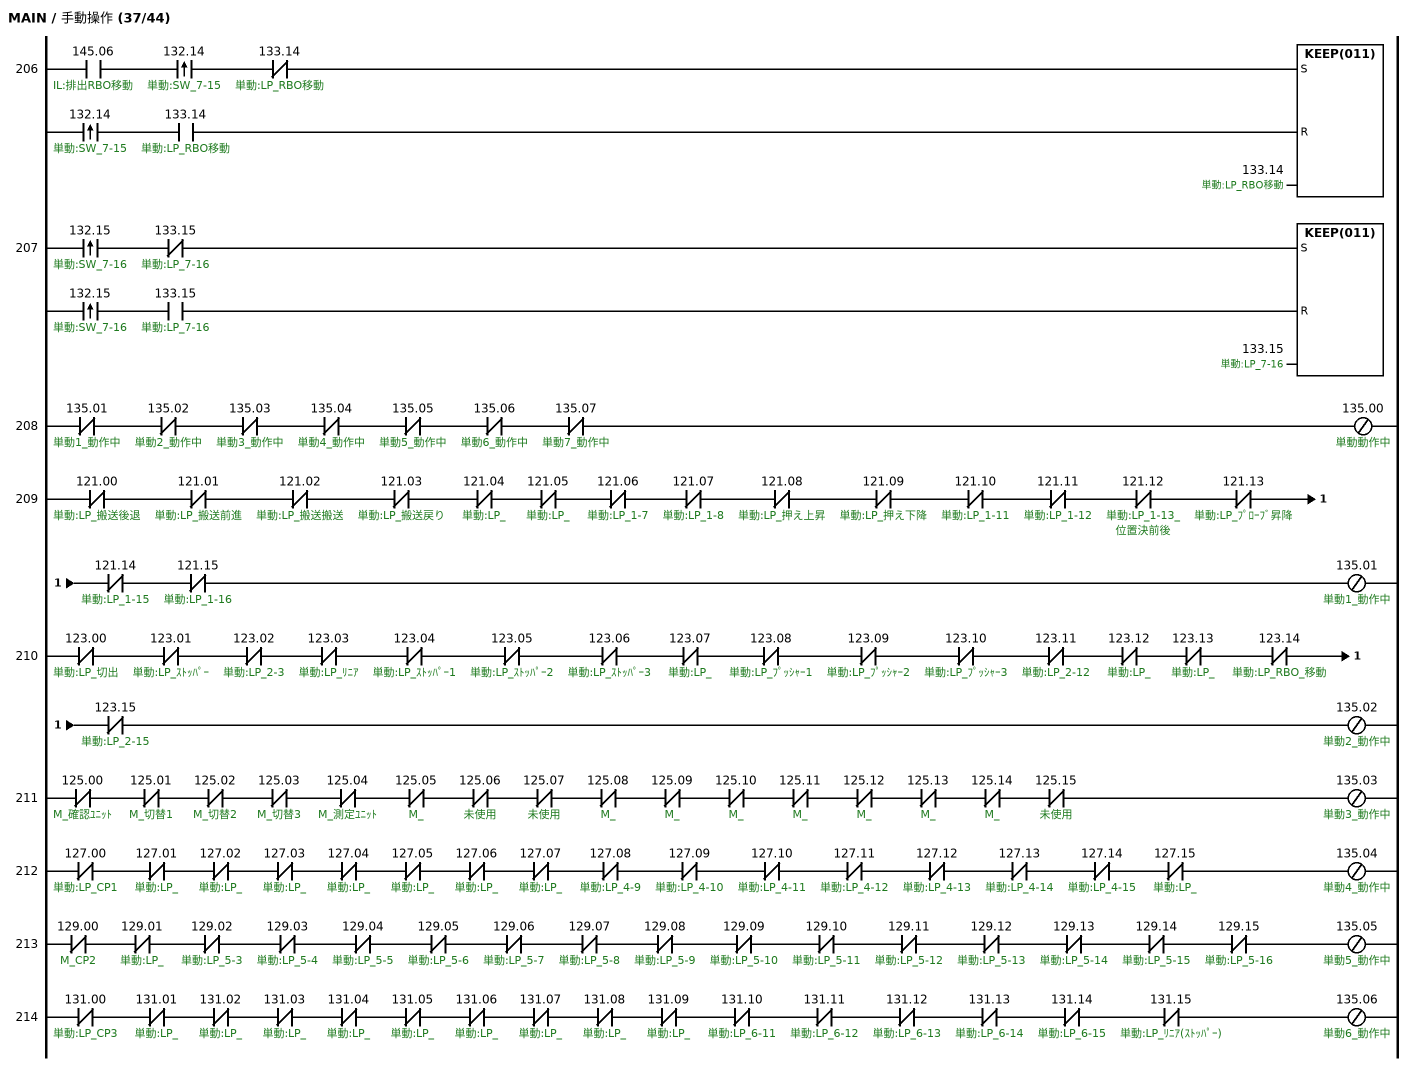
; [picture p72: MAIN / 手動操作, rungs 206-214]
; rung 206
LD 145.06  ; IL:排出RBO移動
@AND 132.14  ; 単動:SW_7-15
ANDNOT 133.14  ; 単動:LP_RBO移動
@LD 132.14  ; 単動:SW_7-15
AND 133.14  ; 単動:LP_RBO移動
KEEP(011) 133.14  ; 単動:LP_RBO移動
; rung 207
@LD 132.15  ; 単動:SW_7-16
ANDNOT 133.15  ; 単動:LP_7-16
@LD 132.15  ; 単動:SW_7-16
AND 133.15  ; 単動:LP_7-16
KEEP(011) 133.15  ; 単動:LP_7-16
; rung 208
LDNOT 135.01  ; 単動1_動作中
ANDNOT 135.02  ; 単動2_動作中
ANDNOT 135.03  ; 単動3_動作中
ANDNOT 135.04  ; 単動4_動作中
ANDNOT 135.05  ; 単動5_動作中
ANDNOT 135.06  ; 単動6_動作中
ANDNOT 135.07  ; 単動7_動作中
OUTNOT 135.00  ; 単動動作中
; rung 209
LDNOT 121.00  ; 単動:LP_搬送後退
ANDNOT 121.01  ; 単動:LP_搬送前進
ANDNOT 121.02  ; 単動:LP_搬送搬送
ANDNOT 121.03  ; 単動:LP_搬送戻り
ANDNOT 121.04  ; 単動:LP_
ANDNOT 121.05  ; 単動:LP_
ANDNOT 121.06  ; 単動:LP_1-7
ANDNOT 121.07  ; 単動:LP_1-8
ANDNOT 121.08  ; 単動:LP_押え上昇
ANDNOT 121.09  ; 単動:LP_押え下降
ANDNOT 121.10  ; 単動:LP_1-11
ANDNOT 121.11  ; 単動:LP_1-12
ANDNOT 121.12  ; 単動:LP_1-13_位置決前後
ANDNOT 121.13  ; 単動:LP_ﾌﾟﾛｰﾌﾞ昇降
ANDNOT 121.14  ; 単動:LP_1-15
ANDNOT 121.15  ; 単動:LP_1-16
OUTNOT 135.01  ; 単動1_動作中
; rung 210
LDNOT 123.00  ; 単動:LP_切出
ANDNOT 123.01  ; 単動:LP_ｽﾄｯﾊﾟｰ
ANDNOT 123.02  ; 単動:LP_2-3
ANDNOT 123.03  ; 単動:LP_ﾘﾆｱ
ANDNOT 123.04  ; 単動:LP_ｽﾄｯﾊﾟｰ1
ANDNOT 123.05  ; 単動:LP_ｽﾄｯﾊﾟｰ2
ANDNOT 123.06  ; 単動:LP_ｽﾄｯﾊﾟｰ3
ANDNOT 123.07  ; 単動:LP_
ANDNOT 123.08  ; 単動:LP_ﾌﾟｯｼｬｰ1
ANDNOT 123.09  ; 単動:LP_ﾌﾟｯｼｬｰ2
ANDNOT 123.10  ; 単動:LP_ﾌﾟｯｼｬｰ3
ANDNOT 123.11  ; 単動:LP_2-12
ANDNOT 123.12  ; 単動:LP_
ANDNOT 123.13  ; 単動:LP_
ANDNOT 123.14  ; 単動:LP_RBO_移動
ANDNOT 123.15  ; 単動:LP_2-15
OUTNOT 135.02  ; 単動2_動作中
; rung 211
LDNOT 125.00  ; M_確認ﾕﾆｯﾄ
ANDNOT 125.01  ; M_切替1
ANDNOT 125.02  ; M_切替2
ANDNOT 125.03  ; M_切替3
ANDNOT 125.04  ; M_測定ﾕﾆｯﾄ
ANDNOT 125.05  ; M_
ANDNOT 125.06  ; 未使用
ANDNOT 125.07  ; 未使用
ANDNOT 125.08  ; M_
ANDNOT 125.09  ; M_
ANDNOT 125.10  ; M_
ANDNOT 125.11  ; M_
ANDNOT 125.12  ; M_
ANDNOT 125.13  ; M_
ANDNOT 125.14  ; M_
ANDNOT 125.15  ; 未使用
OUTNOT 135.03  ; 単動3_動作中
; rung 212
LDNOT 127.00  ; 単動:LP_CP1
ANDNOT 127.01  ; 単動:LP_
ANDNOT 127.02  ; 単動:LP_
ANDNOT 127.03  ; 単動:LP_
ANDNOT 127.04  ; 単動:LP_
ANDNOT 127.05  ; 単動:LP_
ANDNOT 127.06  ; 単動:LP_
ANDNOT 127.07  ; 単動:LP_
ANDNOT 127.08  ; 単動:LP_4-9
ANDNOT 127.09  ; 単動:LP_4-10
ANDNOT 127.10  ; 単動:LP_4-11
ANDNOT 127.11  ; 単動:LP_4-12
ANDNOT 127.12  ; 単動:LP_4-13
ANDNOT 127.13  ; 単動:LP_4-14
ANDNOT 127.14  ; 単動:LP_4-15
ANDNOT 127.15  ; 単動:LP_
OUTNOT 135.04  ; 単動4_動作中
; rung 213
LDNOT 129.00  ; M_CP2
ANDNOT 129.01  ; 単動:LP_
ANDNOT 129.02  ; 単動:LP_5-3
ANDNOT 129.03  ; 単動:LP_5-4
ANDNOT 129.04  ; 単動:LP_5-5
ANDNOT 129.05  ; 単動:LP_5-6
ANDNOT 129.06  ; 単動:LP_5-7
ANDNOT 129.07  ; 単動:LP_5-8
ANDNOT 129.08  ; 単動:LP_5-9
ANDNOT 129.09  ; 単動:LP_5-10
ANDNOT 129.10  ; 単動:LP_5-11
ANDNOT 129.11  ; 単動:LP_5-12
ANDNOT 129.12  ; 単動:LP_5-13
ANDNOT 129.13  ; 単動:LP_5-14
ANDNOT 129.14  ; 単動:LP_5-15
ANDNOT 129.15  ; 単動:LP_5-16
OUTNOT 135.05  ; 単動5_動作中
; rung 214
LDNOT 131.00  ; 単動:LP_CP3
ANDNOT 131.01  ; 単動:LP_
ANDNOT 131.02  ; 単動:LP_
ANDNOT 131.03  ; 単動:LP_
ANDNOT 131.04  ; 単動:LP_
ANDNOT 131.05  ; 単動:LP_
ANDNOT 131.06  ; 単動:LP_
ANDNOT 131.07  ; 単動:LP_
ANDNOT 131.08  ; 単動:LP_
ANDNOT 131.09  ; 単動:LP_
ANDNOT 131.10  ; 単動:LP_6-11
ANDNOT 131.11  ; 単動:LP_6-12
ANDNOT 131.12  ; 単動:LP_6-13
ANDNOT 131.13  ; 単動:LP_6-14
ANDNOT 131.14  ; 単動:LP_6-15
ANDNOT 131.15  ; 単動:LP_ﾘﾆｱ(ｽﾄｯﾊﾟｰ)
OUTNOT 135.06  ; 単動6_動作中

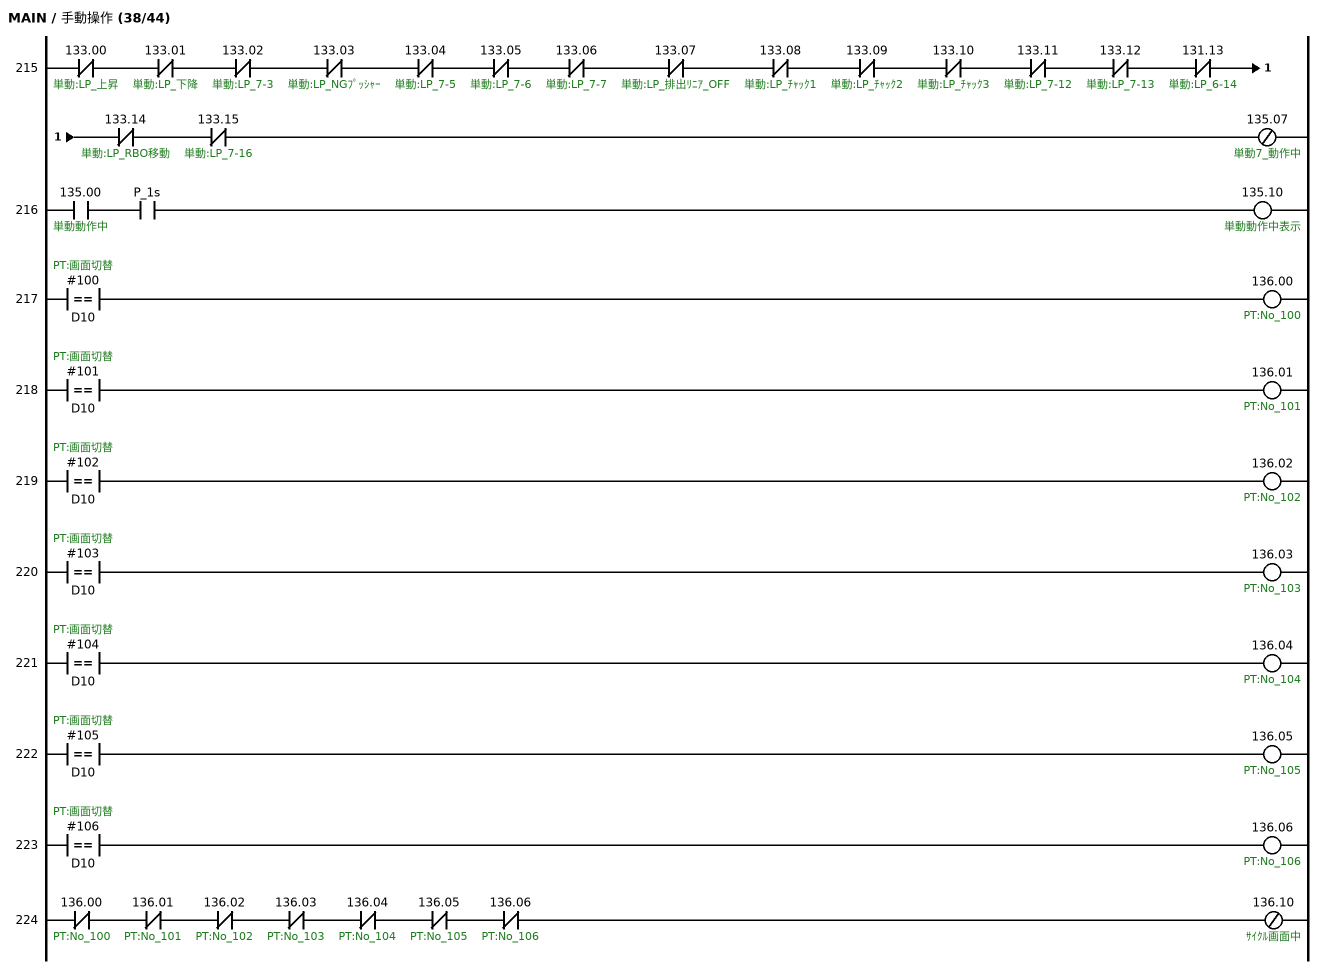
; rung 215
LDNOT 133.00  ; 単動:LP_上昇
ANDNOT 133.01  ; 単動:LP_下降
ANDNOT 133.02  ; 単動:LP_7-3
ANDNOT 133.03  ; 単動:LP_NGﾌﾟｯｼｬｰ
ANDNOT 133.04  ; 単動:LP_7-5
ANDNOT 133.05  ; 単動:LP_7-6
ANDNOT 133.06  ; 単動:LP_7-7
ANDNOT 133.07  ; 単動:LP_排出ﾘﾆｱ_OFF
ANDNOT 133.08  ; 単動:LP_ﾁｬｯｸ1
ANDNOT 133.09  ; 単動:LP_ﾁｬｯｸ2
ANDNOT 133.10  ; 単動:LP_ﾁｬｯｸ3
ANDNOT 133.11  ; 単動:LP_7-12
ANDNOT 133.12  ; 単動:LP_7-13
ANDNOT 131.13  ; 単動:LP_6-14
ANDNOT 133.14  ; 単動:LP_RBO移動
ANDNOT 133.15  ; 単動:LP_7-16
OUTNOT 135.07  ; 単動7_動作中
; rung 216
LD 135.00  ; 単動動作中
AND P_1s
OUT 135.10  ; 単動動作中表示
; rung 217
LD=(300) #100 D10  ; PT:画面切替
OUT 136.00  ; PT:No_100
; rung 218
LD=(300) #101 D10  ; PT:画面切替
OUT 136.01  ; PT:No_101
; rung 219
LD=(300) #102 D10  ; PT:画面切替
OUT 136.02  ; PT:No_102
; rung 220
LD=(300) #103 D10  ; PT:画面切替
OUT 136.03  ; PT:No_103
; rung 221
LD=(300) #104 D10  ; PT:画面切替
OUT 136.04  ; PT:No_104
; rung 222
LD=(300) #105 D10  ; PT:画面切替
OUT 136.05  ; PT:No_105
; rung 223
LD=(300) #106 D10  ; PT:画面切替
OUT 136.06  ; PT:No_106
; rung 224
LDNOT 136.00  ; PT:No_100
ANDNOT 136.01  ; PT:No_101
ANDNOT 136.02  ; PT:No_102
ANDNOT 136.03  ; PT:No_103
ANDNOT 136.04  ; PT:No_104
ANDNOT 136.05  ; PT:No_105
ANDNOT 136.06  ; PT:No_106
OUTNOT 136.10  ; ｻｲｸﾙ画面中

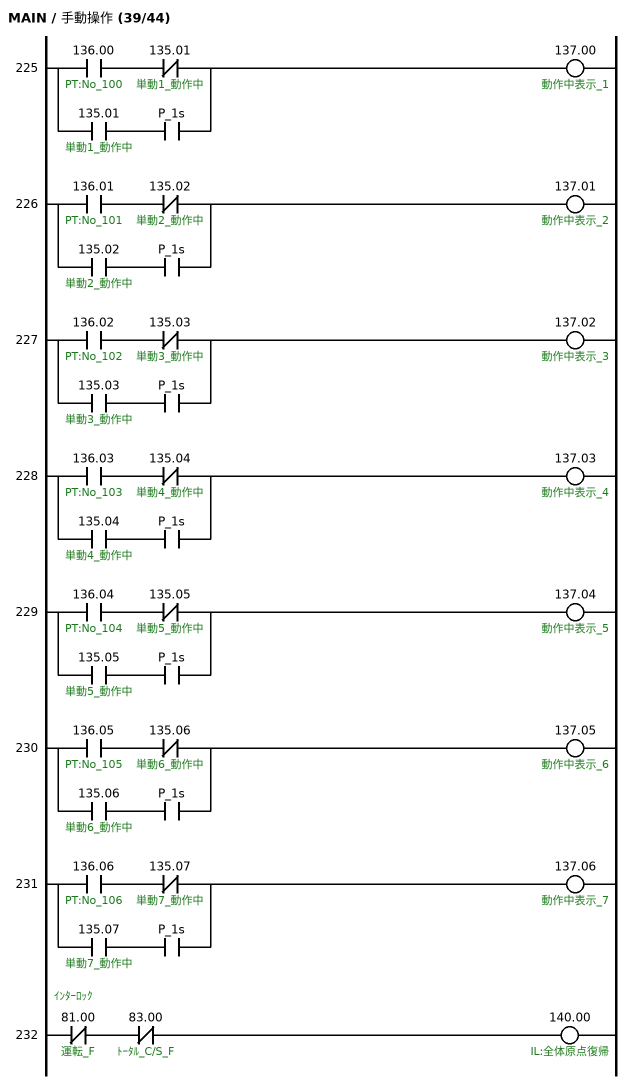
; rung 225
LD 136.00  ; PT:No_100
ANDNOT 135.01  ; 単動1_動作中
LD 135.01  ; 単動1_動作中
AND P_1s
ORLD
OUT 137.00  ; 動作中表示_1
; rung 226
LD 136.01  ; PT:No_101
ANDNOT 135.02  ; 単動2_動作中
LD 135.02  ; 単動2_動作中
AND P_1s
ORLD
OUT 137.01  ; 動作中表示_2
; rung 227
LD 136.02  ; PT:No_102
ANDNOT 135.03  ; 単動3_動作中
LD 135.03  ; 単動3_動作中
AND P_1s
ORLD
OUT 137.02  ; 動作中表示_3
; rung 228
LD 136.03  ; PT:No_103
ANDNOT 135.04  ; 単動4_動作中
LD 135.04  ; 単動4_動作中
AND P_1s
ORLD
OUT 137.03  ; 動作中表示_4
; rung 229
LD 136.04  ; PT:No_104
ANDNOT 135.05  ; 単動5_動作中
LD 135.05  ; 単動5_動作中
AND P_1s
ORLD
OUT 137.04  ; 動作中表示_5
; rung 230
LD 136.05  ; PT:No_105
ANDNOT 135.06  ; 単動6_動作中
LD 135.06  ; 単動6_動作中
AND P_1s
ORLD
OUT 137.05  ; 動作中表示_6
; rung 231
LD 136.06  ; PT:No_106
ANDNOT 135.07  ; 単動7_動作中
LD 135.07  ; 単動7_動作中
AND P_1s
ORLD
OUT 137.06  ; 動作中表示_7
; rung 232: ｲﾝﾀｰﾛｯｸ
LDNOT 81.00  ; 運転_F
ANDNOT 83.00  ; ﾄｰﾀﾙ_C/S_F
OUT 140.00  ; IL:全体原点復帰

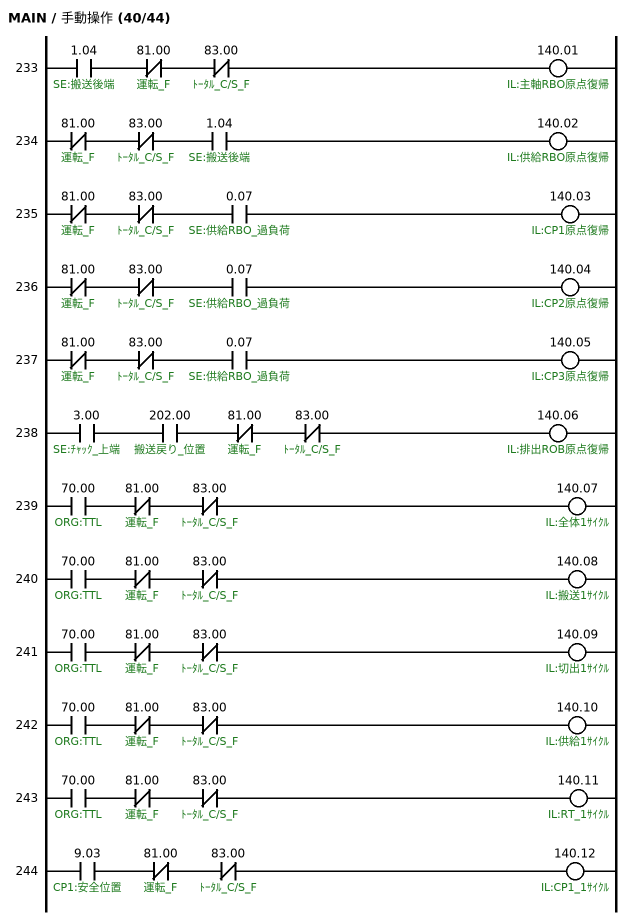
; rung 233
LD 1.04  ; SE:搬送後端
ANDNOT 81.00  ; 運転_F
ANDNOT 83.00  ; ﾄｰﾀﾙ_C/S_F
OUT 140.01  ; IL:主軸RBO原点復帰
; rung 234
LDNOT 81.00  ; 運転_F
ANDNOT 83.00  ; ﾄｰﾀﾙ_C/S_F
AND 1.04  ; SE:搬送後端
OUT 140.02  ; IL:供給RBO原点復帰
; rung 235
LDNOT 81.00  ; 運転_F
ANDNOT 83.00  ; ﾄｰﾀﾙ_C/S_F
AND 0.07  ; SE:供給RBO_過負荷
OUT 140.03  ; IL:CP1原点復帰
; rung 236
LDNOT 81.00  ; 運転_F
ANDNOT 83.00  ; ﾄｰﾀﾙ_C/S_F
AND 0.07  ; SE:供給RBO_過負荷
OUT 140.04  ; IL:CP2原点復帰
; rung 237
LDNOT 81.00  ; 運転_F
ANDNOT 83.00  ; ﾄｰﾀﾙ_C/S_F
AND 0.07  ; SE:供給RBO_過負荷
OUT 140.05  ; IL:CP3原点復帰
; rung 238
LD 3.00  ; SE:ﾁｬｯｸ_上端
AND 202.00  ; 搬送戻り_位置
ANDNOT 81.00  ; 運転_F
ANDNOT 83.00  ; ﾄｰﾀﾙ_C/S_F
OUT 140.06  ; IL:排出ROB原点復帰
; rung 239
LD 70.00  ; ORG:TTL
ANDNOT 81.00  ; 運転_F
ANDNOT 83.00  ; ﾄｰﾀﾙ_C/S_F
OUT 140.07  ; IL:全体1ｻｲｸﾙ
; rung 240
LD 70.00  ; ORG:TTL
ANDNOT 81.00  ; 運転_F
ANDNOT 83.00  ; ﾄｰﾀﾙ_C/S_F
OUT 140.08  ; IL:搬送1ｻｲｸﾙ
; rung 241
LD 70.00  ; ORG:TTL
ANDNOT 81.00  ; 運転_F
ANDNOT 83.00  ; ﾄｰﾀﾙ_C/S_F
OUT 140.09  ; IL:切出1ｻｲｸﾙ
; rung 242
LD 70.00  ; ORG:TTL
ANDNOT 81.00  ; 運転_F
ANDNOT 83.00  ; ﾄｰﾀﾙ_C/S_F
OUT 140.10  ; IL:供給1ｻｲｸﾙ
; rung 243
LD 70.00  ; ORG:TTL
ANDNOT 81.00  ; 運転_F
ANDNOT 83.00  ; ﾄｰﾀﾙ_C/S_F
OUT 140.11  ; IL:RT_1ｻｲｸﾙ
; rung 244
LD 9.03  ; CP1:安全位置
ANDNOT 81.00  ; 運転_F
ANDNOT 83.00  ; ﾄｰﾀﾙ_C/S_F
OUT 140.12  ; IL:CP1_1ｻｲｸﾙ

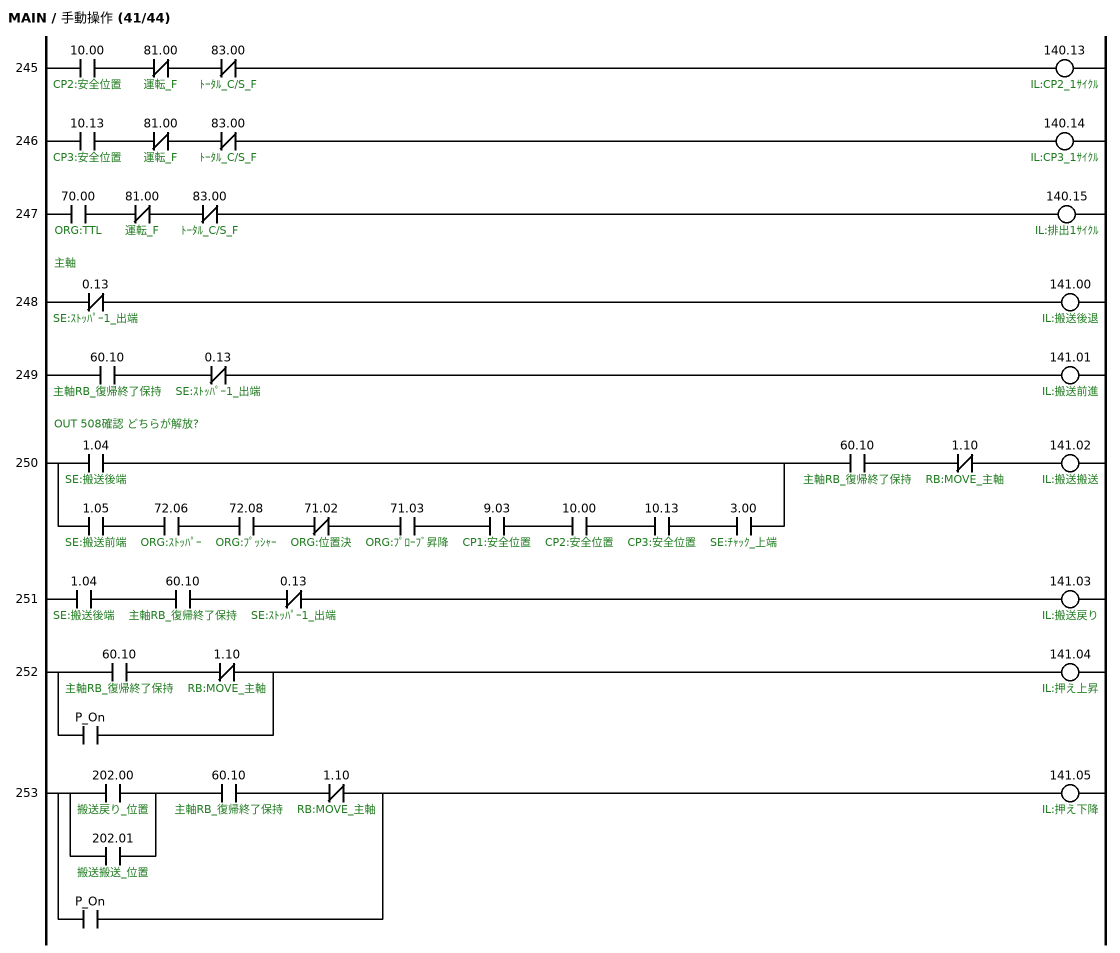
; rung 245
LD 10.00  ; CP2:安全位置
ANDNOT 81.00  ; 運転_F
ANDNOT 83.00  ; ﾄｰﾀﾙ_C/S_F
OUT 140.13  ; IL:CP2_1ｻｲｸﾙ
; rung 246
LD 10.13  ; CP3:安全位置
ANDNOT 81.00  ; 運転_F
ANDNOT 83.00  ; ﾄｰﾀﾙ_C/S_F
OUT 140.14  ; IL:CP3_1ｻｲｸﾙ
; rung 247
LD 70.00  ; ORG:TTL
ANDNOT 81.00  ; 運転_F
ANDNOT 83.00  ; ﾄｰﾀﾙ_C/S_F
OUT 140.15  ; IL:排出1ｻｲｸﾙ
; rung 248: 主軸
LDNOT 0.13  ; SE:ｽﾄｯﾊﾟｰ1_出端
OUT 141.00  ; IL:搬送後退
; rung 249
LD 60.10  ; 主軸RB_復帰終了保持
ANDNOT 0.13  ; SE:ｽﾄｯﾊﾟｰ1_出端
OUT 141.01  ; IL:搬送前進
; rung 250: OUT 508確認 どちらが解放?
LD 1.04  ; SE:搬送後端
LD 1.05  ; SE:搬送前端
AND 72.06  ; ORG:ｽﾄｯﾊﾟｰ
AND 72.08  ; ORG:ﾌﾟｯｼｬｰ
ANDNOT 71.02  ; ORG:位置決
AND 71.03  ; ORG:ﾌﾟﾛｰﾌﾞ昇降
AND 9.03  ; CP1:安全位置
AND 10.00  ; CP2:安全位置
AND 10.13  ; CP3:安全位置
AND 3.00  ; SE:ﾁｬｯｸ_上端
ORLD
AND 60.10  ; 主軸RB_復帰終了保持
ANDNOT 1.10  ; RB:MOVE_主軸
OUT 141.02  ; IL:搬送搬送
; rung 251
LD 1.04  ; SE:搬送後端
AND 60.10  ; 主軸RB_復帰終了保持
ANDNOT 0.13  ; SE:ｽﾄｯﾊﾟｰ1_出端
OUT 141.03  ; IL:搬送戻り
; rung 252
LD 60.10  ; 主軸RB_復帰終了保持
ANDNOT 1.10  ; RB:MOVE_主軸
OR P_On
OUT 141.04  ; IL:押え上昇
; rung 253
LD 202.00  ; 搬送戻り_位置
OR 202.01  ; 搬送搬送_位置
AND 60.10  ; 主軸RB_復帰終了保持
ANDNOT 1.10  ; RB:MOVE_主軸
OR P_On
OUT 141.05  ; IL:押え下降

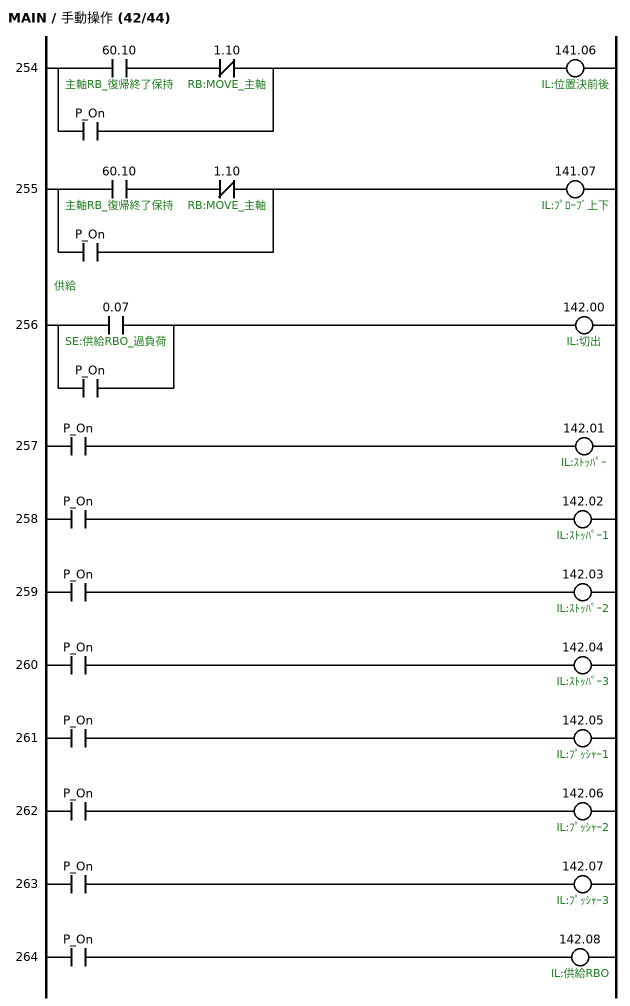
; rung 254
LD 60.10  ; 主軸RB_復帰終了保持
ANDNOT 1.10  ; RB:MOVE_主軸
OR P_On
OUT 141.06  ; IL:位置決前後
; rung 255
LD 60.10  ; 主軸RB_復帰終了保持
ANDNOT 1.10  ; RB:MOVE_主軸
OR P_On
OUT 141.07  ; IL:ﾌﾟﾛｰﾌﾞ上下
; rung 256: 供給
LD 0.07  ; SE:供給RBO_過負荷
OR P_On
OUT 142.00  ; IL:切出
; rung 257
LD P_On
OUT 142.01  ; IL:ｽﾄｯﾊﾟｰ
; rung 258
LD P_On
OUT 142.02  ; IL:ｽﾄｯﾊﾟｰ1
; rung 259
LD P_On
OUT 142.03  ; IL:ｽﾄｯﾊﾟｰ2
; rung 260
LD P_On
OUT 142.04  ; IL:ｽﾄｯﾊﾟｰ3
; rung 261
LD P_On
OUT 142.05  ; IL:ﾌﾟｯｼｬｰ1
; rung 262
LD P_On
OUT 142.06  ; IL:ﾌﾟｯｼｬｰ2
; rung 263
LD P_On
OUT 142.07  ; IL:ﾌﾟｯｼｬｰ3
; rung 264
LD P_On
OUT 142.08  ; IL:供給RBO

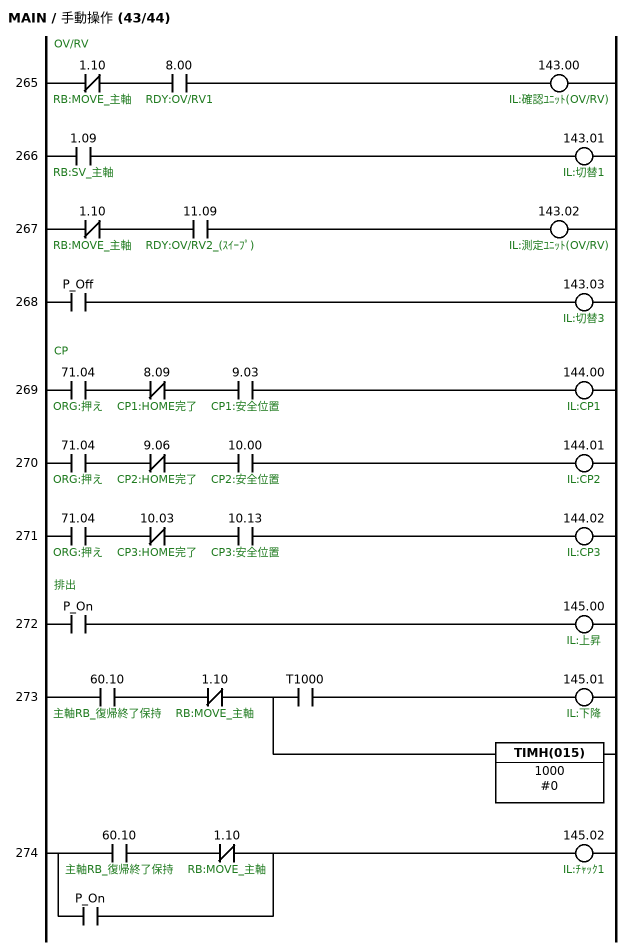
; rung 265: OV/RV
LDNOT 1.10  ; RB:MOVE_主軸
AND 8.00  ; RDY:OV/RV1
OUT 143.00  ; IL:確認ﾕﾆｯﾄ(OV/RV)
; rung 266
LD 1.09  ; RB:SV_主軸
OUT 143.01  ; IL:切替1
; rung 267
LDNOT 1.10  ; RB:MOVE_主軸
AND 11.09  ; RDY:OV/RV2_(ｽｲｰﾌﾟ)
OUT 143.02  ; IL:測定ﾕﾆｯﾄ(OV/RV)
; rung 268
LD P_Off
OUT 143.03  ; IL:切替3
; rung 269: CP
LD 71.04  ; ORG:押え
ANDNOT 8.09  ; CP1:HOME完了
AND 9.03  ; CP1:安全位置
OUT 144.00  ; IL:CP1
; rung 270
LD 71.04  ; ORG:押え
ANDNOT 9.06  ; CP2:HOME完了
AND 10.00  ; CP2:安全位置
OUT 144.01  ; IL:CP2
; rung 271
LD 71.04  ; ORG:押え
ANDNOT 10.03  ; CP3:HOME完了
AND 10.13  ; CP3:安全位置
OUT 144.02  ; IL:CP3
; rung 272: 排出
LD P_On
OUT 145.00  ; IL:上昇
; rung 273
LD 60.10  ; 主軸RB_復帰終了保持
ANDNOT 1.10  ; RB:MOVE_主軸
OUT TR0
AND T1000
OUT 145.01  ; IL:下降
LD TR0
TIMH(015) 1000 #0
; rung 274
LD 60.10  ; 主軸RB_復帰終了保持
ANDNOT 1.10  ; RB:MOVE_主軸
OR P_On
OUT 145.02  ; IL:ﾁｬｯｸ1

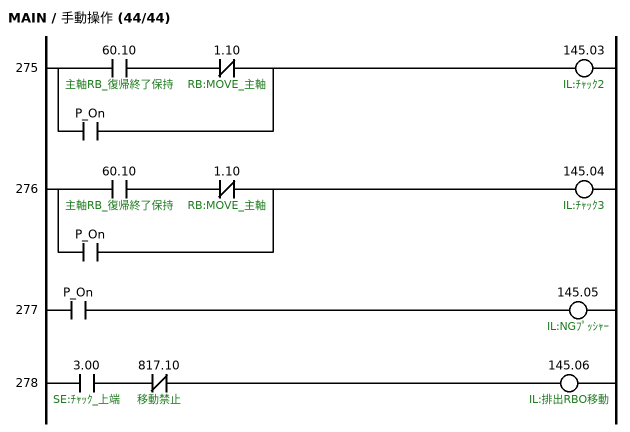
; rung 275
LD 60.10  ; 主軸RB_復帰終了保持
ANDNOT 1.10  ; RB:MOVE_主軸
OR P_On
OUT 145.03  ; IL:ﾁｬｯｸ2
; rung 276
LD 60.10  ; 主軸RB_復帰終了保持
ANDNOT 1.10  ; RB:MOVE_主軸
OR P_On
OUT 145.04  ; IL:ﾁｬｯｸ3
; rung 277
LD P_On
OUT 145.05  ; IL:NGﾌﾟｯｼｬｰ
; rung 278
LD 3.00  ; SE:ﾁｬｯｸ_上端
ANDNOT 817.10  ; 移動禁止
OUT 145.06  ; IL:排出RBO移動

### Section END
; rung 0
END(001)

## Program 主軸 (cyclic task 1)

### Section 動作制御

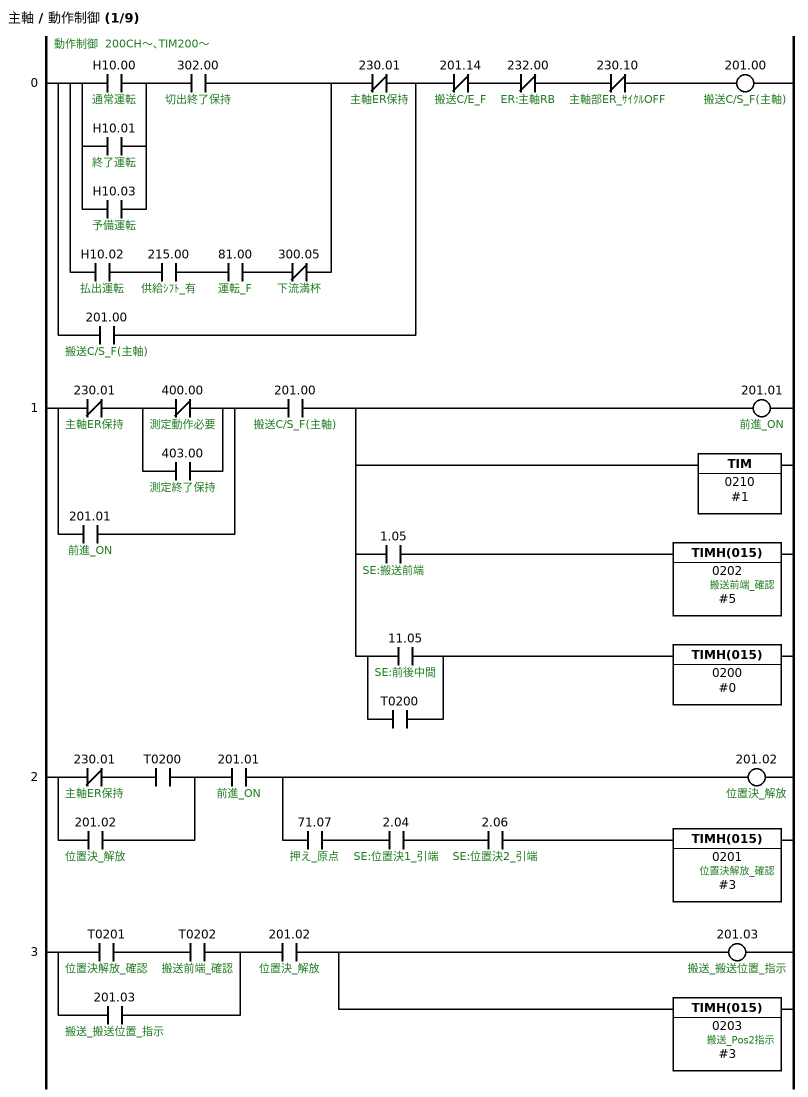
; rung 0: 動作制御  200CH～､TIM200～
LD H10.00  ; 通常運転
OR H10.01  ; 終了運転
OR H10.03  ; 予備運転
AND 302.00  ; 切出終了保持
LD H10.02  ; 払出運転
AND 215.00  ; 供給ｼﾌﾄ_有
AND 81.00  ; 運転_F
ANDNOT 300.05  ; 下流満杯
ORLD
ANDNOT 230.01  ; 主軸ER保持
OR 201.00  ; 搬送C/S_F(主軸)
ANDNOT 201.14  ; 搬送C/E_F
ANDNOT 232.00  ; ER:主軸RB
ANDNOT 230.10  ; 主軸部ER_ｻｲｸﾙOFF
OUT 201.00  ; 搬送C/S_F(主軸)
; rung 1
LDNOT 230.01  ; 主軸ER保持
LDNOT 400.00  ; 測定動作必要
OR 403.00  ; 測定終了保持
ANDLD
OR 201.01  ; 前進_ON
AND 201.00  ; 搬送C/S_F(主軸)
OUT TR0
OUT 201.01  ; 前進_ON
TIM 0210 #1
AND 1.05  ; SE:搬送前端
TIMH(015) 0202 #5  ; 搬送前端_確認
LD TR0
LD 11.05  ; SE:前後中間
OR T0200
ANDLD
TIMH(015) 0200 #0
; rung 2
LDNOT 230.01  ; 主軸ER保持
AND T0200
OR 201.02  ; 位置決_解放
AND 201.01  ; 前進_ON
OUT 201.02  ; 位置決_解放
AND 71.07  ; 押え_原点
AND 2.04  ; SE:位置決1_引端
AND 2.06  ; SE:位置決2_引端
TIMH(015) 0201 #3  ; 位置決解放_確認
; rung 3
LD T0201  ; 位置決解放_確認
AND T0202  ; 搬送前端_確認
OR 201.03  ; 搬送_搬送位置_指示
AND 201.02  ; 位置決_解放
OUT 201.03  ; 搬送_搬送位置_指示
TIMH(015) 0203 #3  ; 搬送_Pos2指示

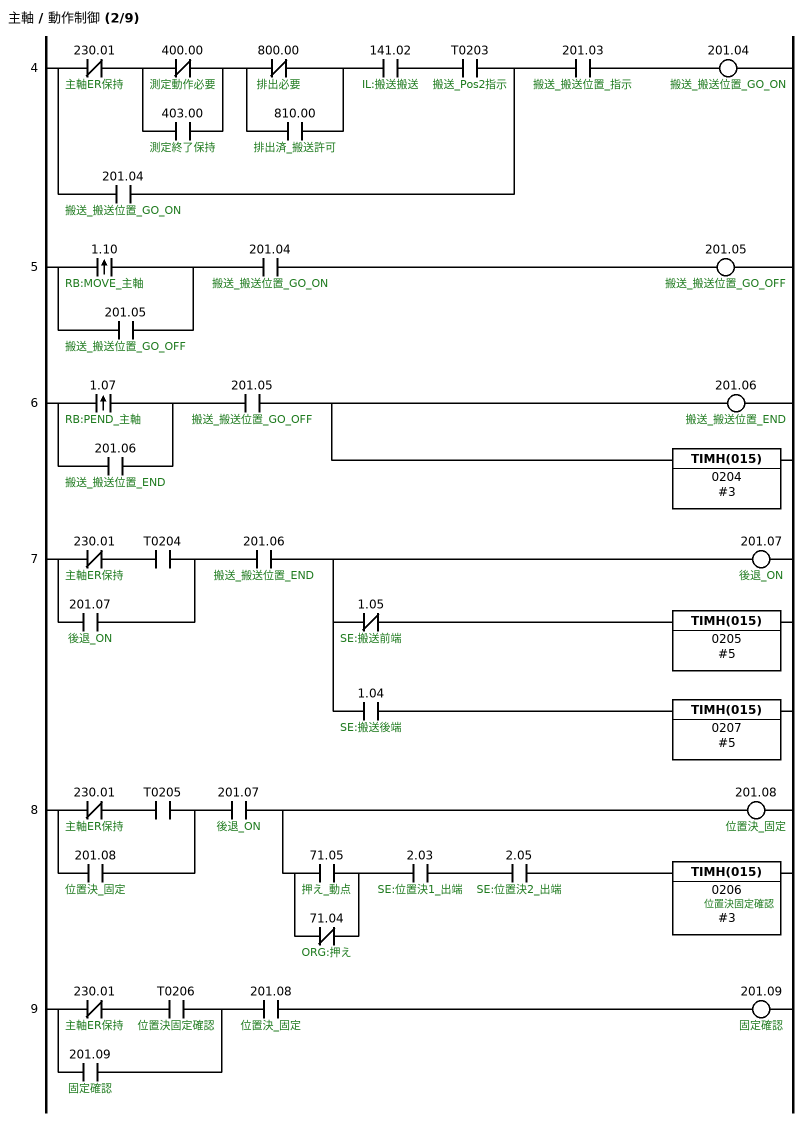
; rung 4
LDNOT 230.01  ; 主軸ER保持
LDNOT 400.00  ; 測定動作必要
OR 403.00  ; 測定終了保持
ANDLD
LDNOT 800.00  ; 排出必要
OR 810.00  ; 排出済_搬送許可
ANDLD
AND 141.02  ; IL:搬送搬送
AND T0203  ; 搬送_Pos2指示
OR 201.04  ; 搬送_搬送位置_GO_ON
AND 201.03  ; 搬送_搬送位置_指示
OUT 201.04  ; 搬送_搬送位置_GO_ON
; rung 5
@LD 1.10  ; RB:MOVE_主軸
OR 201.05  ; 搬送_搬送位置_GO_OFF
AND 201.04  ; 搬送_搬送位置_GO_ON
OUT 201.05  ; 搬送_搬送位置_GO_OFF
; rung 6
@LD 1.07  ; RB:PEND_主軸
OR 201.06  ; 搬送_搬送位置_END
AND 201.05  ; 搬送_搬送位置_GO_OFF
OUT 201.06  ; 搬送_搬送位置_END
TIMH(015) 0204 #3
; rung 7
LDNOT 230.01  ; 主軸ER保持
AND T0204
OR 201.07  ; 後退_ON
AND 201.06  ; 搬送_搬送位置_END
OUT TR0
OUT 201.07  ; 後退_ON
ANDNOT 1.05  ; SE:搬送前端
TIMH(015) 0205 #5
LD TR0
AND 1.04  ; SE:搬送後端
TIMH(015) 0207 #5
; rung 8
LDNOT 230.01  ; 主軸ER保持
AND T0205
OR 201.08  ; 位置決_固定
AND 201.07  ; 後退_ON
OUT 201.08  ; 位置決_固定
LD 71.05  ; 押え_動点
ORNOT 71.04  ; ORG:押え
ANDLD
AND 2.03  ; SE:位置決1_出端
AND 2.05  ; SE:位置決2_出端
TIMH(015) 0206 #3  ; 位置決固定確認
; rung 9
LDNOT 230.01  ; 主軸ER保持
AND T0206  ; 位置決固定確認
OR 201.09  ; 固定確認
AND 201.08  ; 位置決_固定
OUT 201.09  ; 固定確認

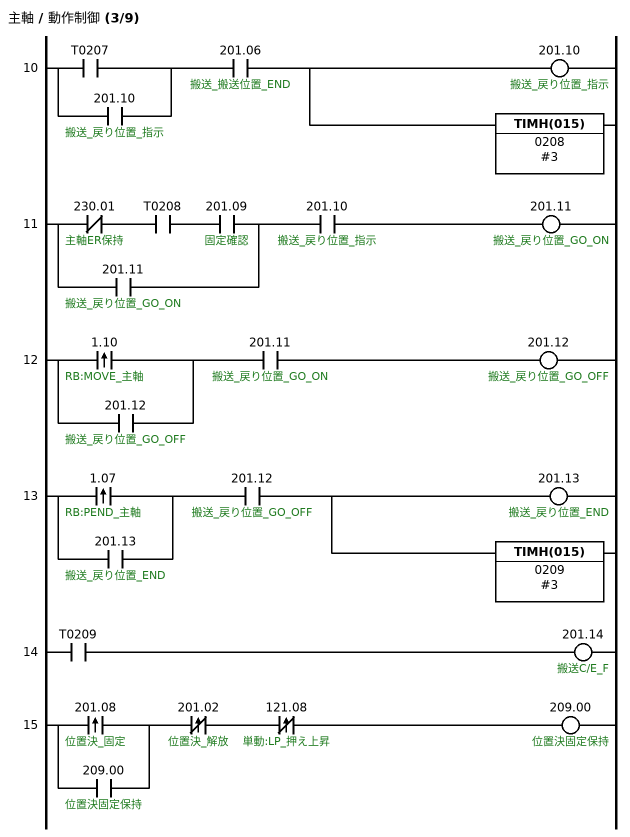
; rung 10
LD T0207
OR 201.10  ; 搬送_戻り位置_指示
AND 201.06  ; 搬送_搬送位置_END
OUT 201.10  ; 搬送_戻り位置_指示
TIMH(015) 0208 #3
; rung 11
LDNOT 230.01  ; 主軸ER保持
AND T0208
AND 201.09  ; 固定確認
OR 201.11  ; 搬送_戻り位置_GO_ON
AND 201.10  ; 搬送_戻り位置_指示
OUT 201.11  ; 搬送_戻り位置_GO_ON
; rung 12
@LD 1.10  ; RB:MOVE_主軸
OR 201.12  ; 搬送_戻り位置_GO_OFF
AND 201.11  ; 搬送_戻り位置_GO_ON
OUT 201.12  ; 搬送_戻り位置_GO_OFF
; rung 13
@LD 1.07  ; RB:PEND_主軸
OR 201.13  ; 搬送_戻り位置_END
AND 201.12  ; 搬送_戻り位置_GO_OFF
OUT 201.13  ; 搬送_戻り位置_END
TIMH(015) 0209 #3
; rung 14
LD T0209
OUT 201.14  ; 搬送C/E_F
; rung 15
@LD 201.08  ; 位置決_固定
OR 209.00  ; 位置決固定保持
@ANDNOT 201.02  ; 位置決_解放
@ANDNOT 121.08  ; 単動:LP_押え上昇
OUT 209.00  ; 位置決固定保持

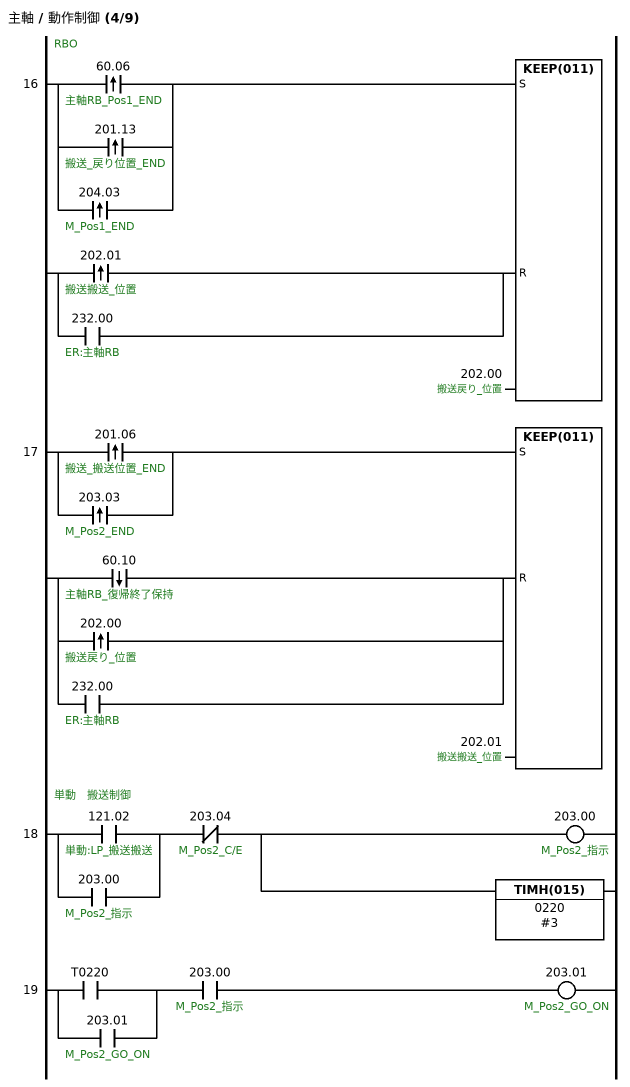
; rung 16: RBO
@LD 60.06  ; 主軸RB_Pos1_END
@OR 201.13  ; 搬送_戻り位置_END
@OR 204.03  ; M_Pos1_END
@LD 202.01  ; 搬送搬送_位置
OR 232.00  ; ER:主軸RB
KEEP(011) 202.00  ; 搬送戻り_位置
; rung 17
@LD 201.06  ; 搬送_搬送位置_END
@OR 203.03  ; M_Pos2_END
%LD 60.10  ; 主軸RB_復帰終了保持
@OR 202.00  ; 搬送戻り_位置
OR 232.00  ; ER:主軸RB
KEEP(011) 202.01  ; 搬送搬送_位置
; rung 18: 単動　搬送制御
LD 121.02  ; 単動:LP_搬送搬送
OR 203.00  ; M_Pos2_指示
ANDNOT 203.04  ; M_Pos2_C/E
OUT 203.00  ; M_Pos2_指示
TIMH(015) 0220 #3
; rung 19
LD T0220
OR 203.01  ; M_Pos2_GO_ON
AND 203.00  ; M_Pos2_指示
OUT 203.01  ; M_Pos2_GO_ON

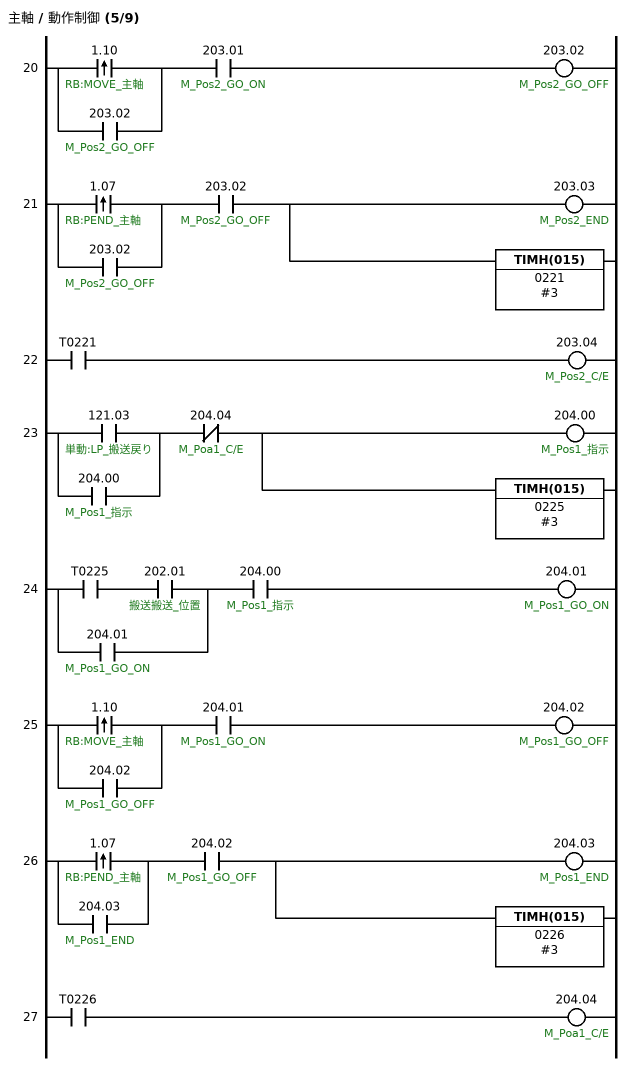
; rung 20
@LD 1.10  ; RB:MOVE_主軸
OR 203.02  ; M_Pos2_GO_OFF
AND 203.01  ; M_Pos2_GO_ON
OUT 203.02  ; M_Pos2_GO_OFF
; rung 21
@LD 1.07  ; RB:PEND_主軸
OR 203.02  ; M_Pos2_GO_OFF
AND 203.02  ; M_Pos2_GO_OFF
OUT 203.03  ; M_Pos2_END
TIMH(015) 0221 #3
; rung 22
LD T0221
OUT 203.04  ; M_Pos2_C/E
; rung 23
LD 121.03  ; 単動:LP_搬送戻り
OR 204.00  ; M_Pos1_指示
ANDNOT 204.04  ; M_Poa1_C/E
OUT 204.00  ; M_Pos1_指示
TIMH(015) 0225 #3
; rung 24
LD T0225
AND 202.01  ; 搬送搬送_位置
OR 204.01  ; M_Pos1_GO_ON
AND 204.00  ; M_Pos1_指示
OUT 204.01  ; M_Pos1_GO_ON
; rung 25
@LD 1.10  ; RB:MOVE_主軸
OR 204.02  ; M_Pos1_GO_OFF
AND 204.01  ; M_Pos1_GO_ON
OUT 204.02  ; M_Pos1_GO_OFF
; rung 26
@LD 1.07  ; RB:PEND_主軸
OR 204.03  ; M_Pos1_END
AND 204.02  ; M_Pos1_GO_OFF
OUT 204.03  ; M_Pos1_END
TIMH(015) 0226 #3
; rung 27
LD T0226
OUT 204.04  ; M_Poa1_C/E

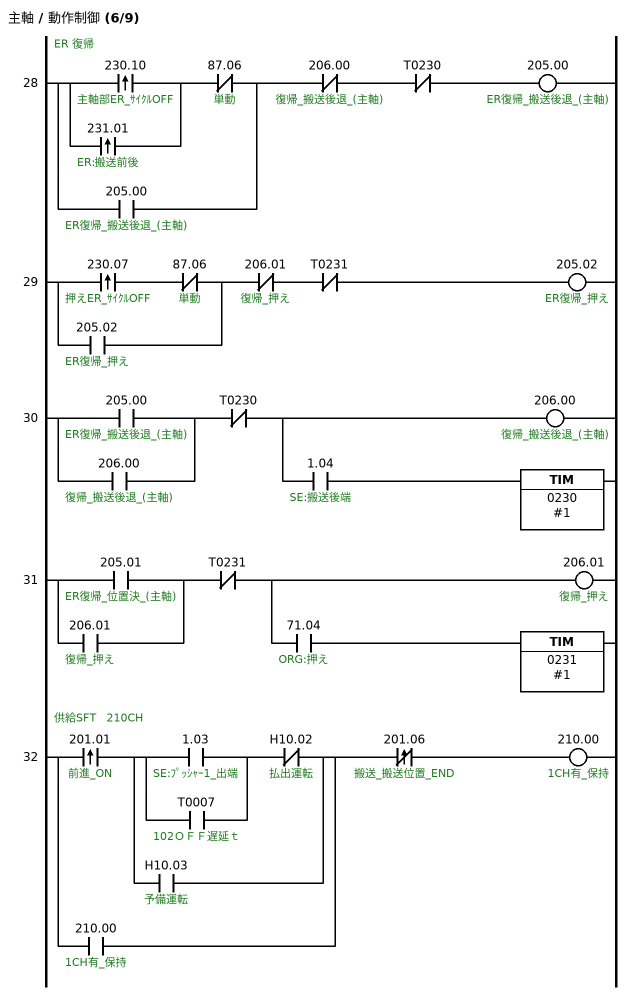
; rung 28: ER 復帰
@LD 230.10  ; 主軸部ER_ｻｲｸﾙOFF
@OR 231.01  ; ER:搬送前後
ANDNOT 87.06  ; 単動
OR 205.00  ; ER復帰_搬送後退_(主軸)
ANDNOT 206.00  ; 復帰_搬送後退_(主軸)
ANDNOT T0230
OUT 205.00  ; ER復帰_搬送後退_(主軸)
; rung 29
@LD 230.07  ; 押えER_ｻｲｸﾙOFF
ANDNOT 87.06  ; 単動
OR 205.02  ; ER復帰_押え
ANDNOT 206.01  ; 復帰_押え
ANDNOT T0231
OUT 205.02  ; ER復帰_押え
; rung 30
LD 205.00  ; ER復帰_搬送後退_(主軸)
OR 206.00  ; 復帰_搬送後退_(主軸)
ANDNOT T0230
OUT 206.00  ; 復帰_搬送後退_(主軸)
AND 1.04  ; SE:搬送後端
TIM 0230 #1
; rung 31
LD 205.01  ; ER復帰_位置決_(主軸)
OR 206.01  ; 復帰_押え
ANDNOT T0231
OUT 206.01  ; 復帰_押え
AND 71.04  ; ORG:押え
TIM 0231 #1
; rung 32: 供給SFT   210CH
@LD 201.01  ; 前進_ON
LD 1.03  ; SE:ﾌﾟｯｼｬｰ1_出端
OR T0007  ; 102ＯＦＦ遅延ｔ
ANDNOT H10.02  ; 払出運転
OR H10.03  ; 予備運転
ANDLD
OR 210.00  ; 1CH有_保持
@ANDNOT 201.06  ; 搬送_搬送位置_END
OUT 210.00  ; 1CH有_保持

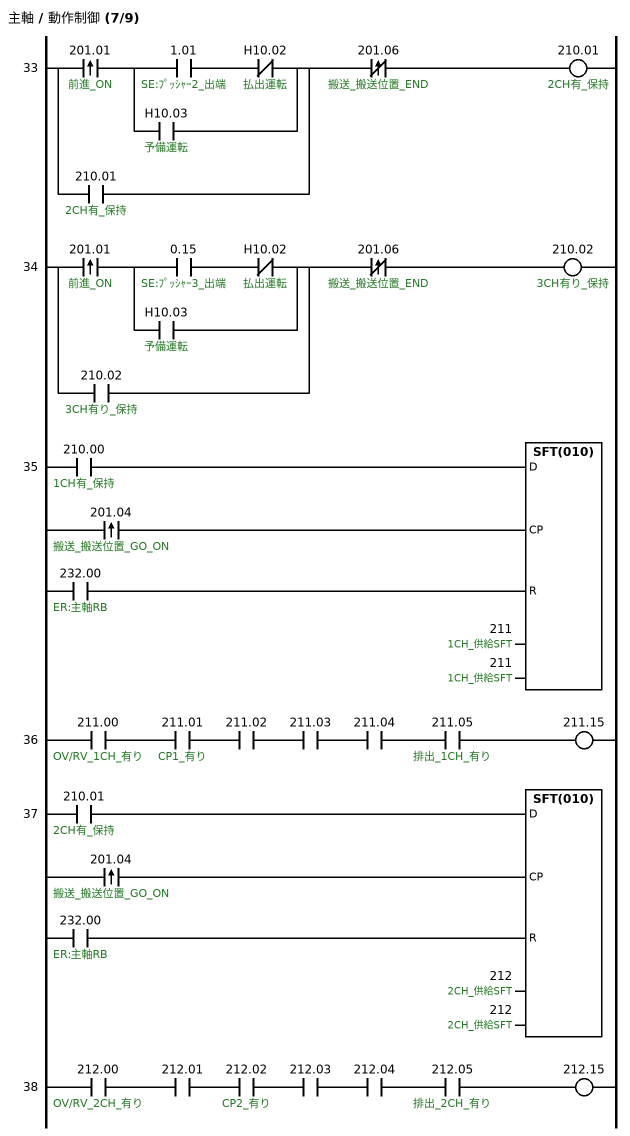
; rung 33
@LD 201.01  ; 前進_ON
LD 1.01  ; SE:ﾌﾟｯｼｬｰ2_出端
ANDNOT H10.02  ; 払出運転
OR H10.03  ; 予備運転
ANDLD
OR 210.01  ; 2CH有_保持
@ANDNOT 201.06  ; 搬送_搬送位置_END
OUT 210.01  ; 2CH有_保持
; rung 34
@LD 201.01  ; 前進_ON
LD 0.15  ; SE:ﾌﾟｯｼｬｰ3_出端
ANDNOT H10.02  ; 払出運転
OR H10.03  ; 予備運転
ANDLD
OR 210.02  ; 3CH有り_保持
@ANDNOT 201.06  ; 搬送_搬送位置_END
OUT 210.02  ; 3CH有り_保持
; rung 35
LD 210.00  ; 1CH有_保持
@LD 201.04  ; 搬送_搬送位置_GO_ON
LD 232.00  ; ER:主軸RB
SFT(010) 211 211  ; 1CH_供給SFT
; rung 36
LD 211.00  ; OV/RV_1CH_有り
AND 211.01  ; CP1_有り
AND 211.02
AND 211.03
AND 211.04
AND 211.05  ; 排出_1CH_有り
OUT 211.15
; rung 37
LD 210.01  ; 2CH有_保持
@LD 201.04  ; 搬送_搬送位置_GO_ON
LD 232.00  ; ER:主軸RB
SFT(010) 212 212  ; 2CH_供給SFT
; rung 38
LD 212.00  ; OV/RV_2CH_有り
AND 212.01
AND 212.02  ; CP2_有り
AND 212.03
AND 212.04
AND 212.05  ; 排出_2CH_有り
OUT 212.15

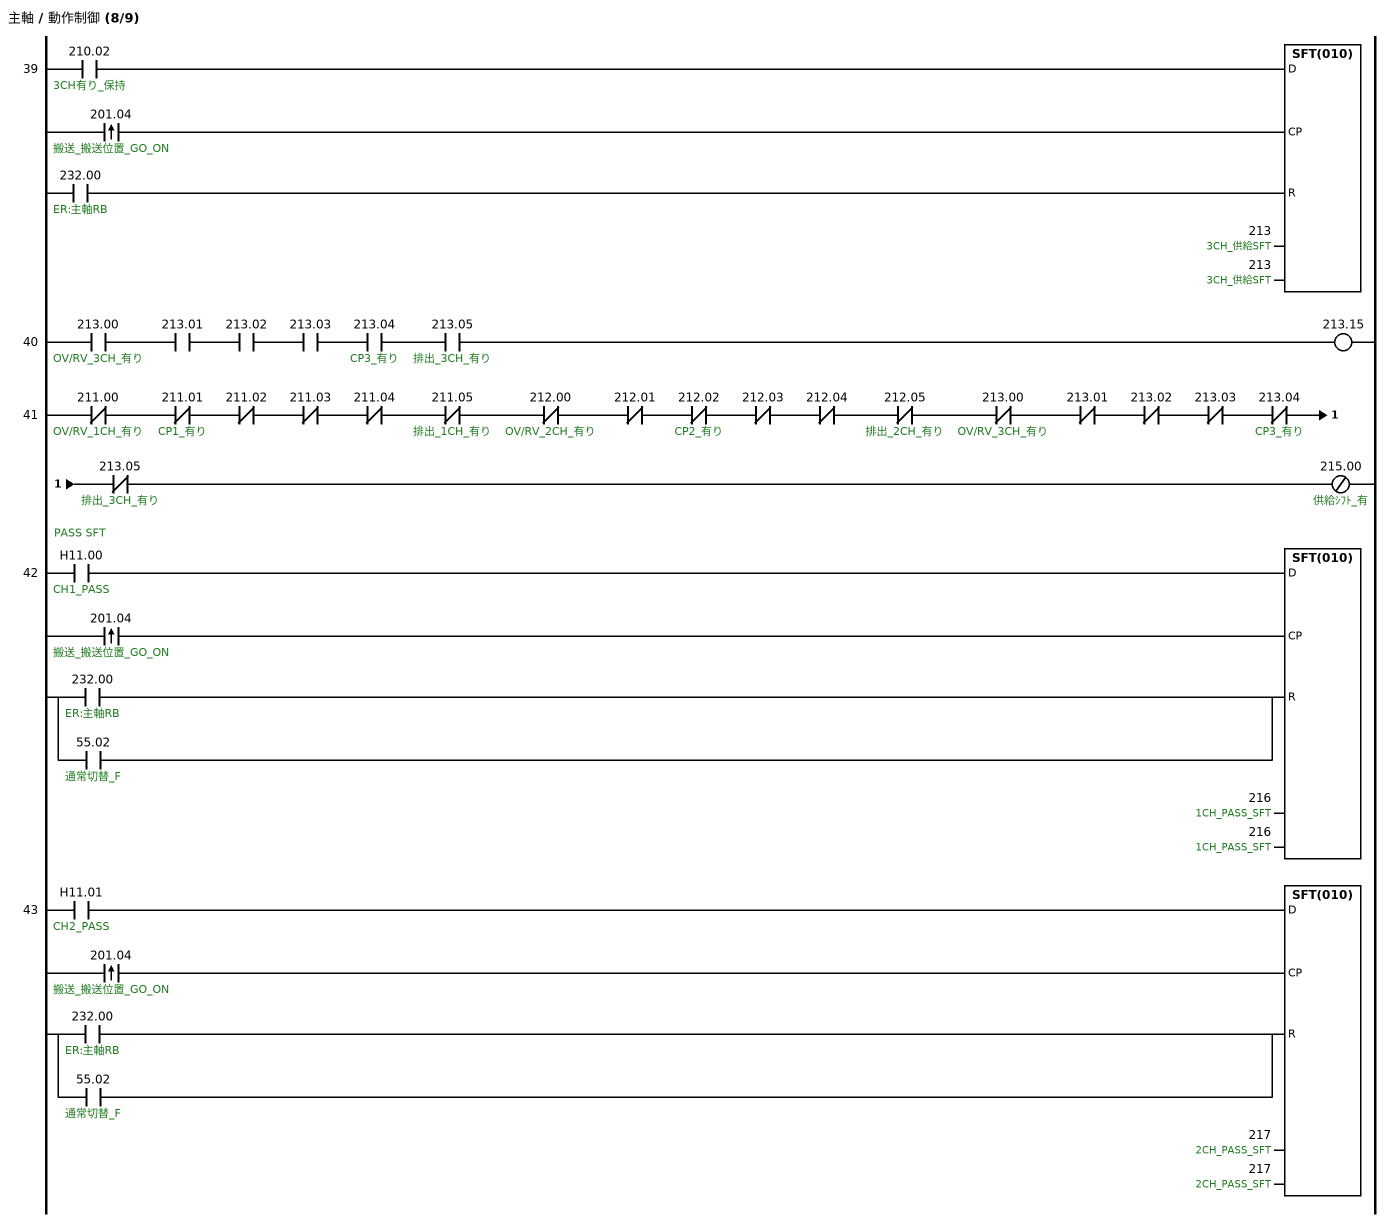
; rung 39
LD 210.02  ; 3CH有り_保持
@LD 201.04  ; 搬送_搬送位置_GO_ON
LD 232.00  ; ER:主軸RB
SFT(010) 213 213  ; 3CH_供給SFT
; rung 40
LD 213.00  ; OV/RV_3CH_有り
AND 213.01
AND 213.02
AND 213.03
AND 213.04  ; CP3_有り
AND 213.05  ; 排出_3CH_有り
OUT 213.15
; rung 41
LDNOT 211.00  ; OV/RV_1CH_有り
ANDNOT 211.01  ; CP1_有り
ANDNOT 211.02
ANDNOT 211.03
ANDNOT 211.04
ANDNOT 211.05  ; 排出_1CH_有り
ANDNOT 212.00  ; OV/RV_2CH_有り
ANDNOT 212.01
ANDNOT 212.02  ; CP2_有り
ANDNOT 212.03
ANDNOT 212.04
ANDNOT 212.05  ; 排出_2CH_有り
ANDNOT 213.00  ; OV/RV_3CH_有り
ANDNOT 213.01
ANDNOT 213.02
ANDNOT 213.03
ANDNOT 213.04  ; CP3_有り
ANDNOT 213.05  ; 排出_3CH_有り
OUTNOT 215.00  ; 供給ｼﾌﾄ_有
; rung 42: PASS SFT
LD H11.00  ; CH1_PASS
@LD 201.04  ; 搬送_搬送位置_GO_ON
LD 232.00  ; ER:主軸RB
OR 55.02  ; 通常切替_F
SFT(010) 216 216  ; 1CH_PASS_SFT
; rung 43
LD H11.01  ; CH2_PASS
@LD 201.04  ; 搬送_搬送位置_GO_ON
LD 232.00  ; ER:主軸RB
OR 55.02  ; 通常切替_F
SFT(010) 217 217  ; 2CH_PASS_SFT

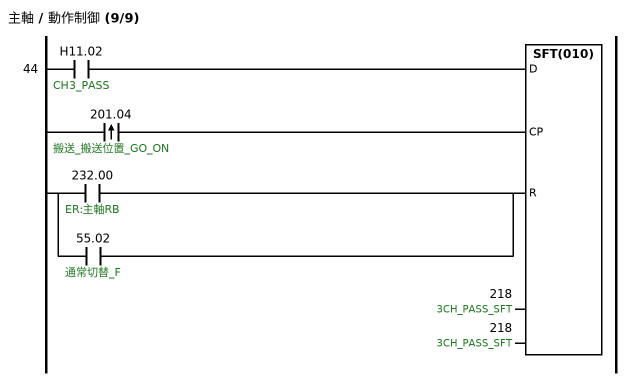
; rung 44
LD H11.02  ; CH3_PASS
@LD 201.04  ; 搬送_搬送位置_GO_ON
LD 232.00  ; ER:主軸RB
OR 55.02  ; 通常切替_F
SFT(010) 218 218  ; 3CH_PASS_SFT

### Section 出力

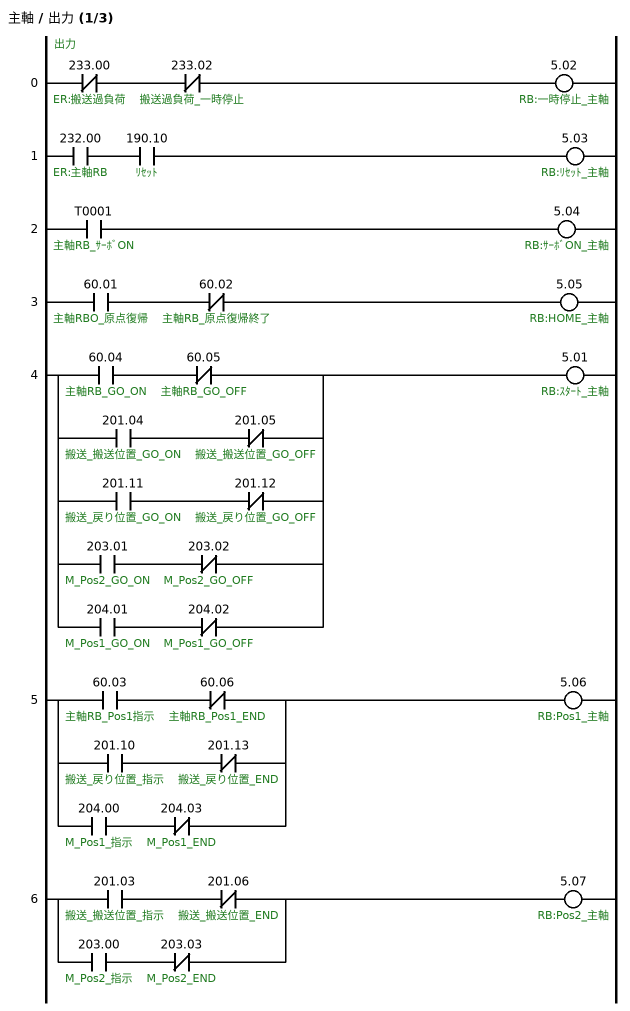
; rung 0: 出力
LDNOT 233.00  ; ER:搬送過負荷
ANDNOT 233.02  ; 搬送過負荷_一時停止
OUT 5.02  ; RB:一時停止_主軸
; rung 1
LD 232.00  ; ER:主軸RB
AND 190.10  ; ﾘｾｯﾄ
OUT 5.03  ; RB:ﾘｾｯﾄ_主軸
; rung 2
LD T0001  ; 主軸RB_ｻｰﾎﾞON
OUT 5.04  ; RB:ｻｰﾎﾞON_主軸
; rung 3
LD 60.01  ; 主軸RBO_原点復帰
ANDNOT 60.02  ; 主軸RB_原点復帰終了
OUT 5.05  ; RB:HOME_主軸
; rung 4
LD 60.04  ; 主軸RB_GO_ON
ANDNOT 60.05  ; 主軸RB_GO_OFF
LD 201.04  ; 搬送_搬送位置_GO_ON
ANDNOT 201.05  ; 搬送_搬送位置_GO_OFF
ORLD
LD 201.11  ; 搬送_戻り位置_GO_ON
ANDNOT 201.12  ; 搬送_戻り位置_GO_OFF
ORLD
LD 203.01  ; M_Pos2_GO_ON
ANDNOT 203.02  ; M_Pos2_GO_OFF
ORLD
LD 204.01  ; M_Pos1_GO_ON
ANDNOT 204.02  ; M_Pos1_GO_OFF
ORLD
OUT 5.01  ; RB:ｽﾀｰﾄ_主軸
; rung 5
LD 60.03  ; 主軸RB_Pos1指示
ANDNOT 60.06  ; 主軸RB_Pos1_END
LD 201.10  ; 搬送_戻り位置_指示
ANDNOT 201.13  ; 搬送_戻り位置_END
ORLD
LD 204.00  ; M_Pos1_指示
ANDNOT 204.03  ; M_Pos1_END
ORLD
OUT 5.06  ; RB:Pos1_主軸
; rung 6
LD 201.03  ; 搬送_搬送位置_指示
ANDNOT 201.06  ; 搬送_搬送位置_END
LD 203.00  ; M_Pos2_指示
ANDNOT 203.03  ; M_Pos2_END
ORLD
OUT 5.07  ; RB:Pos2_主軸

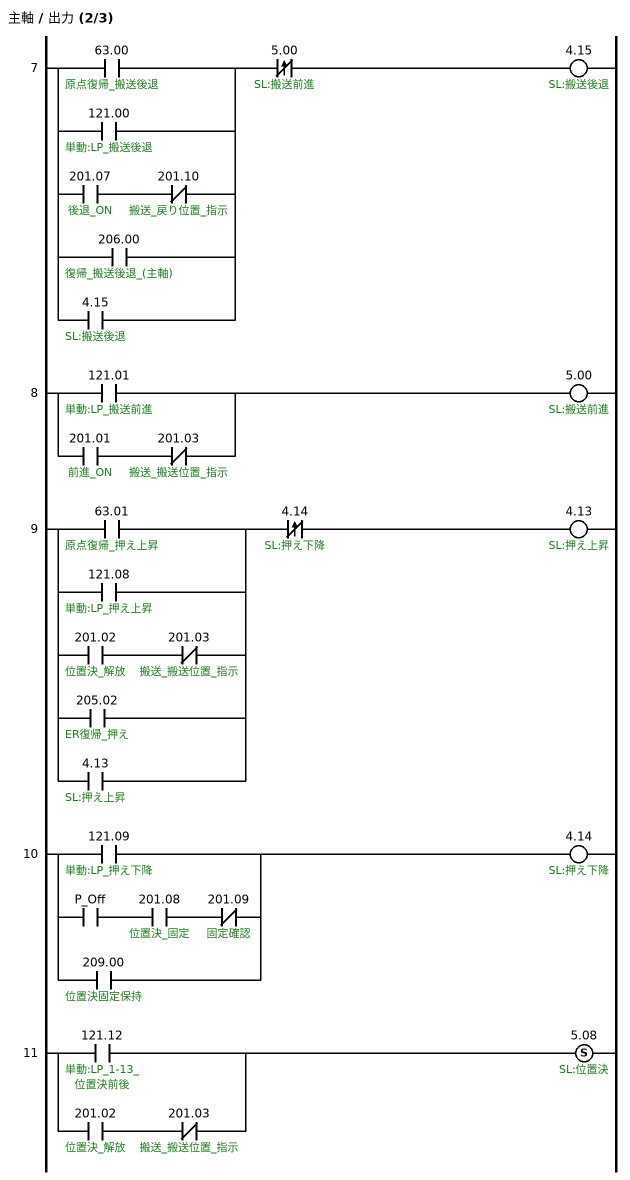
; rung 7
LD 63.00  ; 原点復帰_搬送後退
OR 121.00  ; 単動:LP_搬送後退
LD 201.07  ; 後退_ON
ANDNOT 201.10  ; 搬送_戻り位置_指示
ORLD
OR 206.00  ; 復帰_搬送後退_(主軸)
OR 4.15  ; SL:搬送後退
@ANDNOT 5.00  ; SL:搬送前進
OUT 4.15  ; SL:搬送後退
; rung 8
LD 121.01  ; 単動:LP_搬送前進
LD 201.01  ; 前進_ON
ANDNOT 201.03  ; 搬送_搬送位置_指示
ORLD
OUT 5.00  ; SL:搬送前進
; rung 9
LD 63.01  ; 原点復帰_押え上昇
OR 121.08  ; 単動:LP_押え上昇
LD 201.02  ; 位置決_解放
ANDNOT 201.03  ; 搬送_搬送位置_指示
ORLD
OR 205.02  ; ER復帰_押え
OR 4.13  ; SL:押え上昇
@ANDNOT 4.14  ; SL:押え下降
OUT 4.13  ; SL:押え上昇
; rung 10
LD 121.09  ; 単動:LP_押え下降
LD P_Off
AND 201.08  ; 位置決_固定
ANDNOT 201.09  ; 固定確認
ORLD
OR 209.00  ; 位置決固定保持
OUT 4.14  ; SL:押え下降
; rung 11
LD 121.12  ; 単動:LP_1-13_位置決前後
LD 201.02  ; 位置決_解放
ANDNOT 201.03  ; 搬送_搬送位置_指示
ORLD
SET 5.08  ; SL:位置決

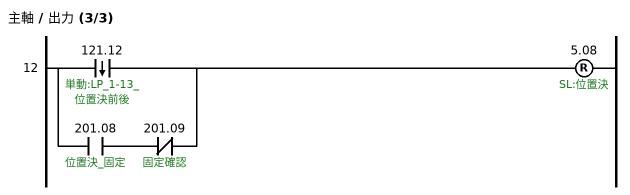
; rung 12
%LD 121.12  ; 単動:LP_1-13_位置決前後
LD 201.08  ; 位置決_固定
ANDNOT 201.09  ; 固定確認
ORLD
RSET 5.08  ; SL:位置決

### Section ｴﾗｰ

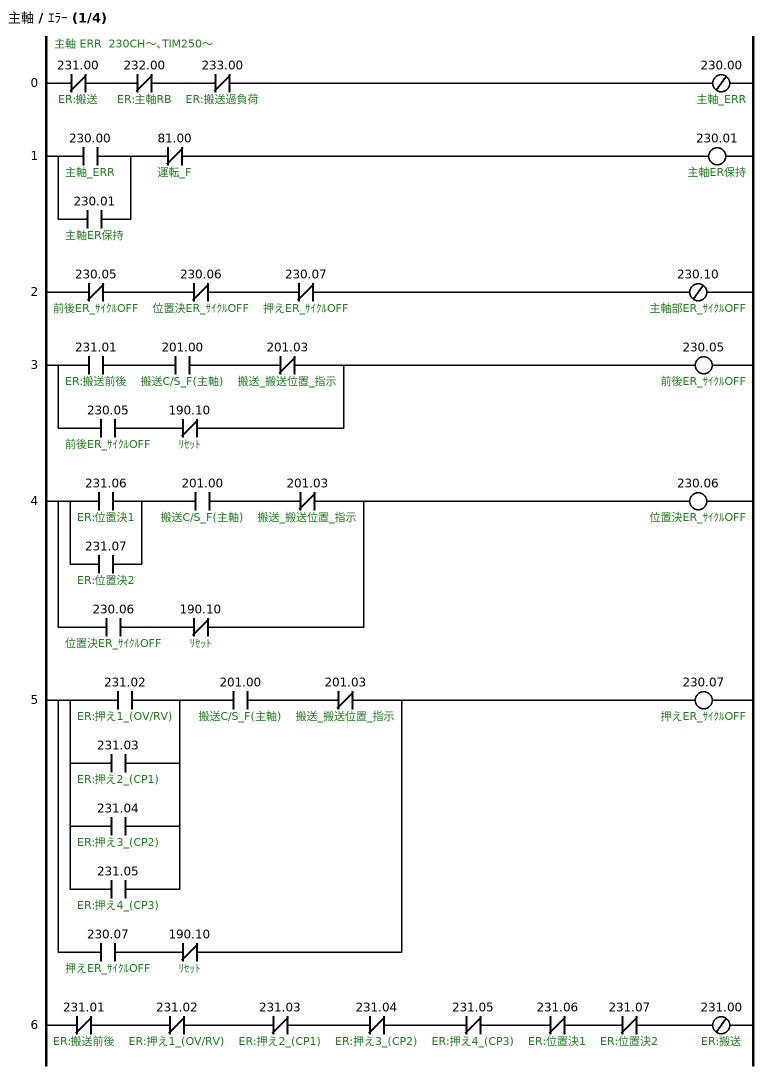
; rung 0: 主軸 ERR  230CH～､TIM250～
LDNOT 231.00  ; ER:搬送
ANDNOT 232.00  ; ER:主軸RB
ANDNOT 233.00  ; ER:搬送過負荷
OUTNOT 230.00  ; 主軸_ERR
; rung 1
LD 230.00  ; 主軸_ERR
OR 230.01  ; 主軸ER保持
ANDNOT 81.00  ; 運転_F
OUT 230.01  ; 主軸ER保持
; rung 2
LDNOT 230.05  ; 前後ER_ｻｲｸﾙOFF
ANDNOT 230.06  ; 位置決ER_ｻｲｸﾙOFF
ANDNOT 230.07  ; 押えER_ｻｲｸﾙOFF
OUTNOT 230.10  ; 主軸部ER_ｻｲｸﾙOFF
; rung 3
LD 231.01  ; ER:搬送前後
AND 201.00  ; 搬送C/S_F(主軸)
ANDNOT 201.03  ; 搬送_搬送位置_指示
LD 230.05  ; 前後ER_ｻｲｸﾙOFF
ANDNOT 190.10  ; ﾘｾｯﾄ
ORLD
OUT 230.05  ; 前後ER_ｻｲｸﾙOFF
; rung 4
LD 231.06  ; ER:位置決1
OR 231.07  ; ER:位置決2
AND 201.00  ; 搬送C/S_F(主軸)
ANDNOT 201.03  ; 搬送_搬送位置_指示
LD 230.06  ; 位置決ER_ｻｲｸﾙOFF
ANDNOT 190.10  ; ﾘｾｯﾄ
ORLD
OUT 230.06  ; 位置決ER_ｻｲｸﾙOFF
; rung 5
LD 231.02  ; ER:押え1_(OV/RV)
OR 231.03  ; ER:押え2_(CP1)
OR 231.04  ; ER:押え3_(CP2)
OR 231.05  ; ER:押え4_(CP3)
AND 201.00  ; 搬送C/S_F(主軸)
ANDNOT 201.03  ; 搬送_搬送位置_指示
LD 230.07  ; 押えER_ｻｲｸﾙOFF
ANDNOT 190.10  ; ﾘｾｯﾄ
ORLD
OUT 230.07  ; 押えER_ｻｲｸﾙOFF
; rung 6
LDNOT 231.01  ; ER:搬送前後
ANDNOT 231.02  ; ER:押え1_(OV/RV)
ANDNOT 231.03  ; ER:押え2_(CP1)
ANDNOT 231.04  ; ER:押え3_(CP2)
ANDNOT 231.05  ; ER:押え4_(CP3)
ANDNOT 231.06  ; ER:位置決1
ANDNOT 231.07  ; ER:位置決2
OUTNOT 231.00  ; ER:搬送

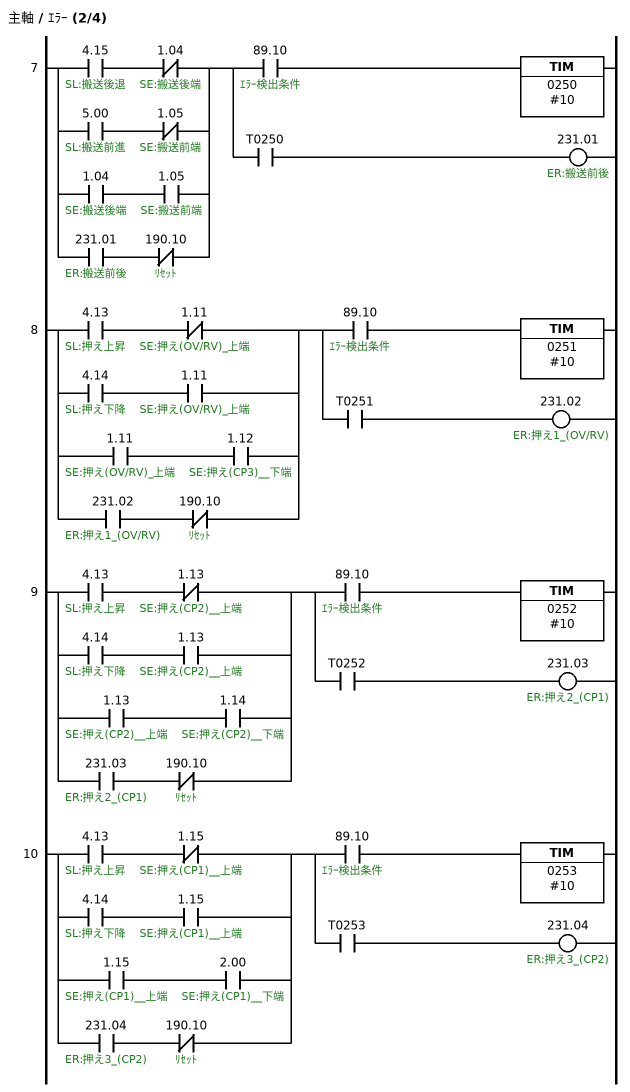
; rung 7
LD 4.15  ; SL:搬送後退
ANDNOT 1.04  ; SE:搬送後端
LD 5.00  ; SL:搬送前進
ANDNOT 1.05  ; SE:搬送前端
ORLD
LD 1.04  ; SE:搬送後端
AND 1.05  ; SE:搬送前端
ORLD
LD 231.01  ; ER:搬送前後
ANDNOT 190.10  ; ﾘｾｯﾄ
ORLD
OUT TR0
AND 89.10  ; ｴﾗｰ検出条件
TIM 0250 #10
LD TR0
AND T0250
OUT 231.01  ; ER:搬送前後
; rung 8
LD 4.13  ; SL:押え上昇
ANDNOT 1.11  ; SE:押え(OV/RV)_上端
LD 4.14  ; SL:押え下降
AND 1.11  ; SE:押え(OV/RV)_上端
ORLD
LD 1.11  ; SE:押え(OV/RV)_上端
AND 1.12  ; SE:押え(CP3)__下端
ORLD
LD 231.02  ; ER:押え1_(OV/RV)
ANDNOT 190.10  ; ﾘｾｯﾄ
ORLD
OUT TR0
AND 89.10  ; ｴﾗｰ検出条件
TIM 0251 #10
LD TR0
AND T0251
OUT 231.02  ; ER:押え1_(OV/RV)
; rung 9
LD 4.13  ; SL:押え上昇
ANDNOT 1.13  ; SE:押え(CP2)__上端
LD 4.14  ; SL:押え下降
AND 1.13  ; SE:押え(CP2)__上端
ORLD
LD 1.13  ; SE:押え(CP2)__上端
AND 1.14  ; SE:押え(CP2)__下端
ORLD
LD 231.03  ; ER:押え2_(CP1)
ANDNOT 190.10  ; ﾘｾｯﾄ
ORLD
OUT TR0
AND 89.10  ; ｴﾗｰ検出条件
TIM 0252 #10
LD TR0
AND T0252
OUT 231.03  ; ER:押え2_(CP1)
; rung 10
LD 4.13  ; SL:押え上昇
ANDNOT 1.15  ; SE:押え(CP1)__上端
LD 4.14  ; SL:押え下降
AND 1.15  ; SE:押え(CP1)__上端
ORLD
LD 1.15  ; SE:押え(CP1)__上端
AND 2.00  ; SE:押え(CP1)__下端
ORLD
LD 231.04  ; ER:押え3_(CP2)
ANDNOT 190.10  ; ﾘｾｯﾄ
ORLD
OUT TR0
AND 89.10  ; ｴﾗｰ検出条件
TIM 0253 #10
LD TR0
AND T0253
OUT 231.04  ; ER:押え3_(CP2)

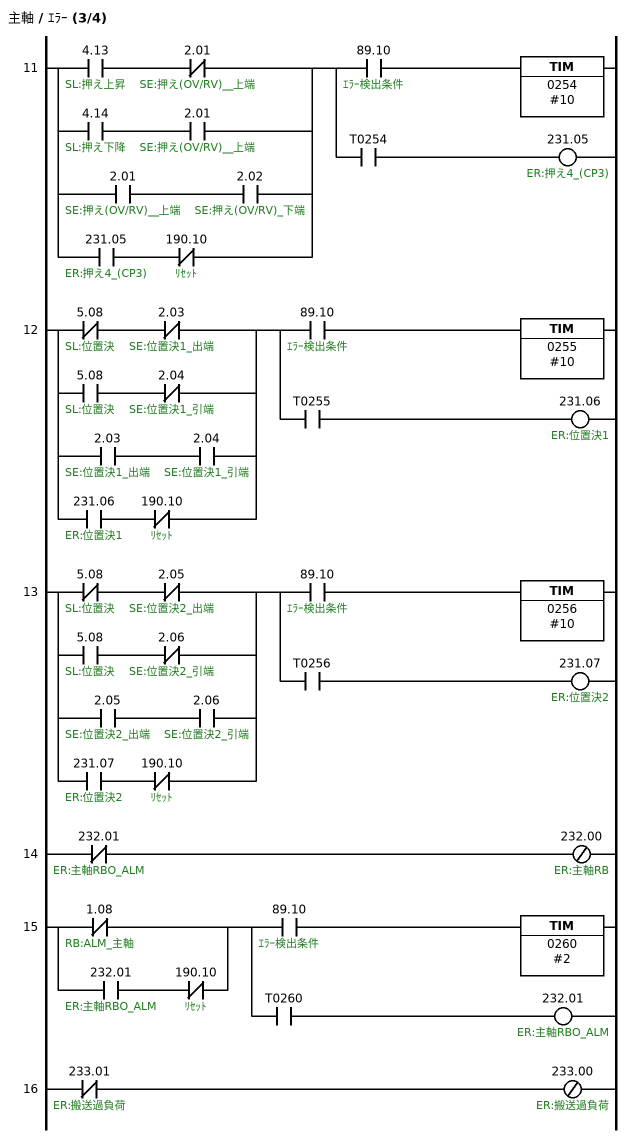
; rung 11
LD 4.13  ; SL:押え上昇
ANDNOT 2.01  ; SE:押え(OV/RV)__上端
LD 4.14  ; SL:押え下降
AND 2.01  ; SE:押え(OV/RV)__上端
ORLD
LD 2.01  ; SE:押え(OV/RV)__上端
AND 2.02  ; SE:押え(OV/RV)_下端
ORLD
LD 231.05  ; ER:押え4_(CP3)
ANDNOT 190.10  ; ﾘｾｯﾄ
ORLD
OUT TR0
AND 89.10  ; ｴﾗｰ検出条件
TIM 0254 #10
LD TR0
AND T0254
OUT 231.05  ; ER:押え4_(CP3)
; rung 12
LDNOT 5.08  ; SL:位置決
ANDNOT 2.03  ; SE:位置決1_出端
LD 5.08  ; SL:位置決
ANDNOT 2.04  ; SE:位置決1_引端
ORLD
LD 2.03  ; SE:位置決1_出端
AND 2.04  ; SE:位置決1_引端
ORLD
LD 231.06  ; ER:位置決1
ANDNOT 190.10  ; ﾘｾｯﾄ
ORLD
OUT TR0
AND 89.10  ; ｴﾗｰ検出条件
TIM 0255 #10
LD TR0
AND T0255
OUT 231.06  ; ER:位置決1
; rung 13
LDNOT 5.08  ; SL:位置決
ANDNOT 2.05  ; SE:位置決2_出端
LD 5.08  ; SL:位置決
ANDNOT 2.06  ; SE:位置決2_引端
ORLD
LD 2.05  ; SE:位置決2_出端
AND 2.06  ; SE:位置決2_引端
ORLD
LD 231.07  ; ER:位置決2
ANDNOT 190.10  ; ﾘｾｯﾄ
ORLD
OUT TR0
AND 89.10  ; ｴﾗｰ検出条件
TIM 0256 #10
LD TR0
AND T0256
OUT 231.07  ; ER:位置決2
; rung 14
LDNOT 232.01  ; ER:主軸RBO_ALM
OUTNOT 232.00  ; ER:主軸RB
; rung 15
LDNOT 1.08  ; RB:ALM_主軸
LD 232.01  ; ER:主軸RBO_ALM
ANDNOT 190.10  ; ﾘｾｯﾄ
ORLD
OUT TR0
AND 89.10  ; ｴﾗｰ検出条件
TIM 0260 #2
LD TR0
AND T0260
OUT 232.01  ; ER:主軸RBO_ALM
; rung 16
LDNOT 233.01  ; ER:搬送過負荷
OUTNOT 233.00  ; ER:搬送過負荷

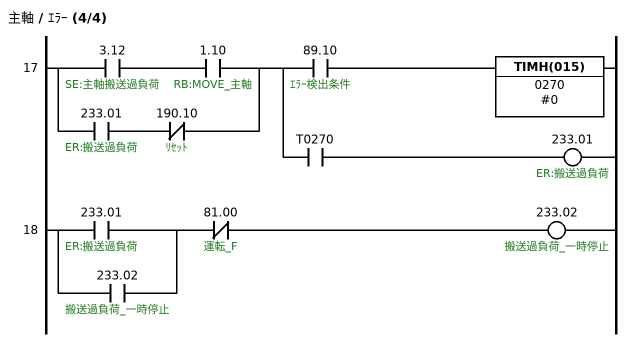
; rung 17
LD 3.12  ; SE:主軸搬送過負荷
AND 1.10  ; RB:MOVE_主軸
LD 233.01  ; ER:搬送過負荷
ANDNOT 190.10  ; ﾘｾｯﾄ
ORLD
OUT TR0
AND 89.10  ; ｴﾗｰ検出条件
TIMH(015) 0270 #0
LD TR0
AND T0270
OUT 233.01  ; ER:搬送過負荷
; rung 18
LD 233.01  ; ER:搬送過負荷
OR 233.02  ; 搬送過負荷_一時停止
ANDNOT 81.00  ; 運転_F
OUT 233.02  ; 搬送過負荷_一時停止

### Section END
; rung 0
END(001)

## Program 供給 (cyclic task 2)

### Section 制御

